TYPE s_DataSampleCav :
STRUCT
	cav : ARRAY[0..8] OF s_DataSamplePocketQty;
END_STRUCT
END_TYPE

(* stored: Version 1.1.0.1, ProductVersion 3.1.4024.11
   DUT s_DataSampleCav: Id {1eb56bfe-f652-4cb5-a8bf-6258cb2f9d08} *)
